Universal Robots PolyScope program: straight top demo.urp

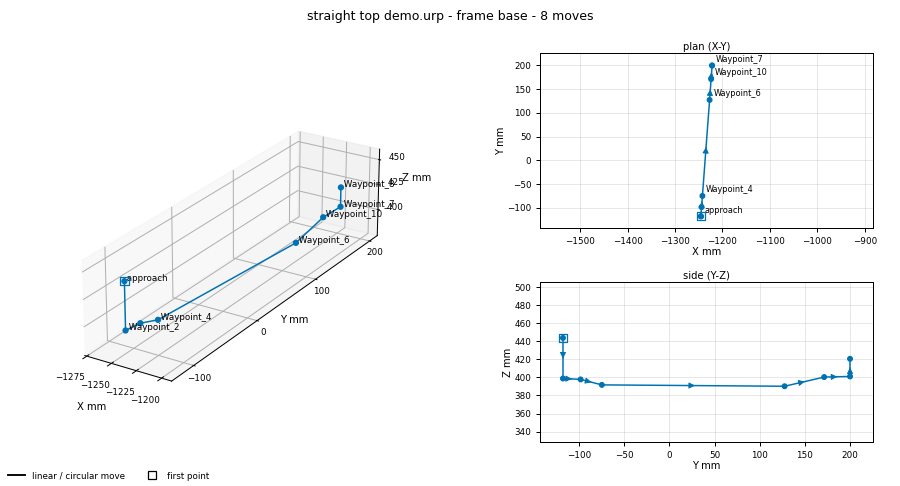
[picture p0: tool path of straight top demo.urp in frame base, 8 of 8 moves have a stored position in this frame; points joined in program order, loops and branches not executed]
Program straight top demo (installation=default directory=/programs createdIn=5.21.3 lastSavedIn=5.21.3 robotSerialNumber=20246801938)
Calibrated DH parameters: a=[-0.000071, -0.790281, -0.600694, 0.000061, -0.000039, 0]; d=[0.236272, 604.465945, 132.116513, -736.382239, 0.159268, 0.154005]; alpha=[1.570254, -0.000567, 0.000559, 1.571709, -1.56999, 0]; deltaTheta=[0, -0.409357, 7.293326, -0.600784, -0.000001, -0.000001]
InitVariablesNode
Robot Program (runOnlyOnce=false)
  Folder demo points
    SuppressedNode
      MoveJ speed 60 deg/s, acceleration 80 deg/s^2 (useActiveTCP=true optimoveEnabled=false optiMoveSpeed=0.3 optiMoveAcceleration=0.09) feature=Base
        Waypoint safepoint: TCP in base x=-924.031 y=-406.135 z=434.478 mm, rx=0.2815 ry=3.1224 rz=-0.0127 rad; joints [20.095, -84.517, 98.026, -13.052, 120.45, 0.706] deg; TCP offset x=-9.5 y=-328 z=105.73 mm, rx=1.2092 ry=-1.2092 rz=1.2092 rad
        Waypoint Waypoint_1: TCP in base x=-1245.427 y=-117.911 z=408.125 mm, rx=0.117 ry=3.1324 rz=-0.0121 rad; joints [-3.268, -71.759, 84.221, -12.093, 91.065, 0.481] deg
    MoveJ speed 60 deg/s, acceleration 80 deg/s^2 (useActiveTCP=true optimoveEnabled=false optiMoveSpeed=0.3 optiMoveAcceleration=0.09) feature=Base
      Waypoint approach: TCP in base x=-1245.427 y=-117.911 z=443.767 mm, rx=0.1153 ry=3.1146 rz=0.2657 rad; joints [0.095, -71.189, 81.089, -9.527, 94.427, -9.693] deg
    SuppressedNode
      MoveL speed 12 mm/s, acceleration 1200 mm/s^2 (useActiveTCP=true optimoveEnabled=false optiMoveSpeed=0.3 optiMoveAcceleration=0.09) feature=Base
        SuppressedNode
          Waypoint approach: TCP in base x=-1245.427 y=-117.911 z=443.767 mm, rx=0.1153 ry=3.1146 rz=0.2657 rad; joints [0.095, -71.189, 81.089, -9.527, 94.427, -9.693] deg
        Waypoint Waypoint_2: TCP in base x=-1245.427 y=-117.911 z=398.812 mm, rx=0.1153 ry=3.1146 rz=0.2657 rad; joints [0.094, -70.583, 83.855, -12.899, 94.427, -9.694] deg
        SuppressedNode
          Waypoint Waypoint_3: TCP in base x=-1245.053 y=-112.838 z=396.452 mm, rx=0.1153 ry=3.1146 rz=0.2657 rad; joints [-0.199, -70.637, 84.122, -13.113, 94.134, -9.696] deg
        SuppressedNode
          Waypoint startofstraight: TCP in base x=-1245.427 y=-117.911 z=392.061 mm, rx=0.117 ry=3.1324 rz=-0.0121 rad; joints [-3.269, -71.517, 85.183, -13.298, 91.065, 0.48] deg
        Waypoint Waypoint_4: TCP in base x=-1242.205 y=-74.854 z=391.739 mm, rx=0.117 ry=3.1324 rz=-0.0121 rad; joints [-5.806, -72.074, 85.979, -13.538, 88.528, 0.464] deg
        Waypoint endofstraight: TCP in base x=-1217.812 y=251.074 z=389.296 mm, rx=0.117 ry=3.1324 rz=-0.0121 rad; joints [-24.861, -72.273, 86.451, -13.802, 69.473, 0.339] deg
        SuppressedNode
          Waypoint tilted: TCP in base x=-1217.812 y=251.074 z=396.846 mm, rx=0.1155 ry=3.1161 rz=0.2513 rad; joints [-21.772, -72.765, 86.984, -13.847, 72.562, -9.303] deg
        Waypoint andmoved: TCP in base x=-1213.76 y=305.753 z=399.277 mm, rx=0.1155 ry=3.1161 rz=0.2513 rad; joints [-24.854, -72.342, 86.209, -13.491, 69.481, -9.324] deg
        Waypoint Waypoint_5: TCP in base x=-1213.76 y=305.753 z=427.713 mm, rx=0.1155 ry=3.1161 rz=0.2513 rad; joints [-24.853, -72.762, 84.487, -11.35, 69.481, -9.323] deg
    SuppressedNode
      MoveL speed 12 mm/s, acceleration 1200 mm/s^2 (useActiveTCP=true optimoveEnabled=false optiMoveSpeed=0.3 optiMoveAcceleration=0.09) feature=Base
        SuppressedNode
          Waypoint approach: TCP in base x=-1245.427 y=-117.911 z=443.767 mm, rx=0.1153 ry=3.1146 rz=0.2657 rad; joints [0.095, -71.189, 81.089, -9.527, 94.427, -9.693] deg
        Waypoint Waypoint_2: TCP in base x=-1245.427 y=-117.911 z=398.812 mm, rx=0.1153 ry=3.1146 rz=0.2657 rad; joints [0.094, -70.583, 83.855, -12.899, 94.427, -9.694] deg
        SuppressedNode
          Waypoint Waypoint_3: TCP in base x=-1245.053 y=-112.838 z=396.452 mm, rx=0.1153 ry=3.1146 rz=0.2657 rad; joints [-0.199, -70.637, 84.122, -13.113, 94.134, -9.696] deg
        SuppressedNode
          Waypoint startofstraight: TCP in base x=-1245.427 y=-117.911 z=392.061 mm, rx=0.117 ry=3.1324 rz=-0.0121 rad; joints [-3.269, -71.517, 85.183, -13.298, 91.065, 0.48] deg
        Waypoint Waypoint_4: TCP in base x=-1242.205 y=-74.854 z=391.739 mm, rx=0.117 ry=3.1324 rz=-0.0121 rad; joints [-5.806, -72.074, 85.979, -13.538, 88.528, 0.464] deg
        Waypoint Waypoint_6: TCP in base x=-1227.078 y=127.461 z=390.228 mm, rx=0.117 ry=3.1324 rz=-0.0121 rad; joints [-17.792, -73.042, 87.423, -14.014, 76.541, 0.387] deg
        Waypoint Waypoint_7: TCP in base x=-1221.788 y=199.927 z=401.073 mm, rx=0.1148 ry=3.1059 rz=0.3369 rad; joints [-17.791, -73.052, 87.345, -13.917, 76.545, -12.44] deg
        Waypoint Waypoint_8: TCP in base x=-1221.788 y=199.927 z=420.619 mm, rx=0.1148 ry=3.1059 rz=0.3369 rad; joints [-17.79, -73.357, 86.175, -12.443, 76.545, -12.44] deg
        SuppressedNode
          Waypoint tilted: TCP in base x=-1217.812 y=251.074 z=396.846 mm, rx=0.1155 ry=3.1161 rz=0.2513 rad; joints [-21.772, -72.765, 86.984, -13.847, 72.562, -9.303] deg
        SuppressedNode
          Waypoint andmoved: TCP in base x=-1213.76 y=305.753 z=399.277 mm, rx=0.1155 ry=3.1161 rz=0.2513 rad; joints [-24.854, -72.342, 86.209, -13.491, 69.481, -9.324] deg
        SuppressedNode
          Waypoint Waypoint_5: TCP in base x=-1213.76 y=305.753 z=427.713 mm, rx=0.1155 ry=3.1161 rz=0.2513 rad; joints [-24.853, -72.762, 84.487, -11.35, 69.481, -9.323] deg
    MoveL speed 12 mm/s, acceleration 1200 mm/s^2 (useActiveTCP=true optimoveEnabled=false optiMoveSpeed=0.3 optiMoveAcceleration=0.09) feature=Base
      SuppressedNode
        Waypoint approach: TCP in base x=-1245.427 y=-117.911 z=443.767 mm, rx=0.1153 ry=3.1146 rz=0.2657 rad; joints [0.095, -71.189, 81.089, -9.527, 94.427, -9.693] deg
      Waypoint Waypoint_2: TCP in base x=-1245.427 y=-117.911 z=398.812 mm, rx=0.1153 ry=3.1146 rz=0.2657 rad; joints [0.094, -70.583, 83.855, -12.899, 94.427, -9.694] deg
      Wait Sleep waitTime=4
      URCap WireTank Serial (WireTank Serial, WireTank, LLC) dataModel(NODE_TITLE=ur1, byte_array=true, Command=[100,0,0], OUTPUT_ENTRY=Static)
      Wait Sleep waitTime=1
      Waypoint Waypoint_9: TCP in base x=-1243.99 y=-98.373 z=397.795 mm, rx=0.1153 ry=3.1146 rz=0.2657 rad; joints [-1.036, -70.908, 84.392, -13.113, 93.297, -9.702] deg
      SuppressedNode
        Waypoint Waypoint_3: TCP in base x=-1245.053 y=-112.838 z=396.452 mm, rx=0.1153 ry=3.1146 rz=0.2657 rad; joints [-0.199, -70.637, 84.122, -13.113, 94.134, -9.696] deg
      SuppressedNode
        Waypoint startofstraight: TCP in base x=-1245.427 y=-117.911 z=392.061 mm, rx=0.117 ry=3.1324 rz=-0.0121 rad; joints [-3.269, -71.517, 85.183, -13.298, 91.065, 0.48] deg
      Waypoint Waypoint_4: TCP in base x=-1242.205 y=-74.854 z=391.739 mm, rx=0.117 ry=3.1324 rz=-0.0121 rad; joints [-5.806, -72.074, 85.979, -13.538, 88.528, 0.464] deg
      Waypoint Waypoint_6: TCP in base x=-1227.078 y=127.461 z=390.228 mm, rx=0.117 ry=3.1324 rz=-0.0121 rad; joints [-17.792, -73.042, 87.423, -14.014, 76.541, 0.387] deg
      Waypoint Waypoint_10: TCP in base x=-1223.883 y=171.298 z=400.392 mm, rx=0.1148 ry=3.1059 rz=0.3369 rad; joints [-16.112, -73.071, 87.426, -13.981, 78.224, -12.429] deg
      URCap WireTank Serial (WireTank Serial, WireTank, LLC) dataModel(NODE_TITLE=ur1, byte_array=true, Command=[100,0,0], OUTPUT_ENTRY=Static)
      Waypoint Waypoint_7: TCP in base x=-1221.788 y=199.927 z=401.073 mm, rx=0.1148 ry=3.1059 rz=0.3369 rad; joints [-17.791, -73.052, 87.345, -13.917, 76.545, -12.44] deg
      Wait Sleep waitTime=1
      Waypoint Waypoint_8: TCP in base x=-1221.788 y=199.927 z=420.619 mm, rx=0.1148 ry=3.1059 rz=0.3369 rad; joints [-17.79, -73.357, 86.175, -12.443, 76.545, -12.44] deg
      SuppressedNode
        Waypoint tilted: TCP in base x=-1217.812 y=251.074 z=396.846 mm, rx=0.1155 ry=3.1161 rz=0.2513 rad; joints [-21.772, -72.765, 86.984, -13.847, 72.562, -9.303] deg
      SuppressedNode
        Waypoint andmoved: TCP in base x=-1213.76 y=305.753 z=399.277 mm, rx=0.1155 ry=3.1161 rz=0.2513 rad; joints [-24.854, -72.342, 86.209, -13.491, 69.481, -9.324] deg
      SuppressedNode
        Waypoint Waypoint_5: TCP in base x=-1213.76 y=305.753 z=427.713 mm, rx=0.1155 ry=3.1161 rz=0.2513 rad; joints [-24.853, -72.762, 84.487, -11.35, 69.481, -9.323] deg
